{attribute 'qualified_only'}
{attribute 'global_init_slot' := '40520'}
VAR_GLOBAL
	fbSilownik								: FB_Silownik_Kontola (		fbCzujnikPozycja0 			:= GVL_Wejscia_IO.bCzujnik0S1, 
																		fbCzujnikPozycjaMax 		:= GVL_Wejscia_IO.bCzujnikMaxS1,
																		fbElektrozawor 				:= GVL_Wyjscia_IO.fbElektrozaworS1);
	fbSilownik1								: FB_Silownik_Kontola (		fbCzujnikPozycja0 			:= GVL_Wejscia_IO.bCzujnik0S2, 
																		fbCzujnikPozycjaMax 		:= GVL_Wejscia_IO.bCzujnikMaxS2,
																		fbElektrozawor 				:= GVL_Wyjscia_IO.fbElektrozaworS2);																
	fbPrzesuwacz							: FB_PrzesuwaczNaSilowniku (bCzujnik0Zabieraka			:= GVL_Wejscia_IO.bCzujnik0Z,
		                                                                bCzujnikMaxZabieraka		:= GVL_Wejscia_IO.bCzujnikMaxZ	,
	                                                                    fbElektrozaworZabieraka		:= GVL_Wyjscia_IO.fbElektrozaworZ,
	                                                                    bCzujnik0Przesuwacza		:= GVL_Wejscia_IO.bCzujnik0P,
	                                                                    bCzujnikMaxPrzesuwacza		:= GVL_Wejscia_IO.bCzujnikMaxP	,
	                                                                    fbElektrozaworPrzesuwacza	:= GVL_Wyjscia_IO.fbElektrozaworP);
END_VAR

(* stored: Version 1.1.0.1, ProductVersion 3.1.4024.11
   GVL GVL_Elementy: Id {79604a35-f506-4d38-acf4-c8c8ed6f71ed} *)
